{attribute addProperty BoxType "AT2050-0501-0017"}
{attribute addProperty Id "A_0088_AT2050_5501_0017_AT2050_5501AT2050_3DCFC8D064080"}
{attribute addProperty CRC "2205315928"}
{attribute addProperty SizeInBites "640"}
{attribute addProperty SizeInBytes "80"}
TYPE A_0056_AT2050_0501_0017_83727358 EXTENDS AT2050_9506A482 :
STRUCT
	{attribute addProperty Name "A_0088_AT2050_5501_0017_AT2050_5501"}
	A_0088_AT2050_5501_0017_AT2050_5501 : AT2050_3DCFC8D0;
END_STRUCT
END_TYPE

(* stored: Version 1.2.0.0, ProductVersion 3.1.4024.9
   DUT A_0056_AT2050_0501_0017_83727358: Id {c23b512a-05ca-4691-9826-53751638bde6} *)
